(* Logix 5000 project; controller cal1615 1756-L62 rev 20.11; software revision 20.05; part 23 of 82 *)
(* tags used below, declared in another part *)
   FAULT : BOOL;   // Fault AFI
   HMI : BOOL;   // AFI HMI
   p01_sys_scp : SYS_SCP;   // System Scaling
   p01r02 : routine;   // System Misc Control
   p01r09_pb_global_reset : BOOL;   // System Modes PB: Global Fault Reset
   p12_ai_exhaust_amps : REAL;   // Zone 2 Analog Input Exhaust Fan Amps
   p12_ai_exhaust_hz : REAL;   // Zone 2 Analog Input Exhaust Fan HZ
   p12_ai_exhaust_hz_max : REAL;   // Zone 2 Analog Input Exhaust Fan Max HZ
   p12_ai_exhaust_rpm : REAL;   // Zone 2 Analog Input Exhaust Fan RPM
   p12_ai_lfl : REAL;   // Zone 2 Analog Input Lower Flash Limit
   p12_ai_prs : REAL;   // Zone 2 Analog Input Pressure
   p12_ai_recirc_amps : REAL;   // Zone 2 Analog Input Recirc Fan Amps
   p12_ai_recirc_hz : REAL;   // Zone 2 Analog Input Supply Fan HZ
   p12_ai_recirc_hz_max : REAL;   // Zone 2 Analog Input Supply Fan Max HZ
   p12_ai_recirc_rpm : REAL;   // Zone 2 Analog Input Recirc Fan RPM
   p12_ai_tc01 : REAL;   // Zone 2 Analog Input Control Thermocouple 1
   p12_ai_tc02 : REAL;   // Zone 2 Analog Input Control Thermocouple 2
   p12_ao_cv : REAL;   // Zone 2 Analog Output Control Valve
   p12_ao_exhaust_selected_speed : REAL;   // Zone 2 Analog Output Exhaust Fan VFD Selected Speed
   p12_ao_recirc_selected_speed : REAL;   // Zone 2 Analog Output Recirc Fan VFD Selected Speed
   p12_di_burner_auto : BOOL;   // Zone 2 Digital Input Burner Auto
   p12_di_burner_safeties_ok : BOOL;   // Zone 2 Digital Input Burner Safeties Ok
   p12_di_door_open : BOOL;   // Zone 2 Digital Input Access Door Open
   p12_di_exh : acs800_di_normal;   // Zone 2 Digital Inputs Exhaust Fan
   p12_di_exh_fan_mtr_ts : BOOL;   // Zone 2 Digital Input Exhaust Fan Motor Thermostat OK
   p12_di_exh_flow_ok : BOOL;   // Zone 2 Digital Input Exhaust Flow OK
   p12_di_flame_failure : BOOL;   // Zone 2 Digital Input Flame Failure
   p12_di_flame_on : BOOL;   // Zone 2 Digital Input Burner is On
   p12_di_fresh_air_clean : BOOL;   // Zone 2 Digital Input Fresh Air Filter Dirty
   p12_di_high_limit_temp_ok : BOOL;   // Zone 2 Digital Input High Limit Temperature OK
   p12_di_recirc : acs800_di_normal;   // Zone 2 Digital Inputs Recirc Fan
   p12_di_recirc_fan_mtr_ts : BOOL;   // Zone 2 Digital Input Recirc Fan Motor Thermostat OK
   p12_di_recirc_flow_ok : BOOL;   // Zone 2 Digital Input Recirc Flow OK
   p12_di_sp0 : BOOL;
   p12_di_sp00 : BOOL;   // Zone 2 Digital Input Combustion Blower Pressure OK
   p12_di_sp1 : BOOL;
   p12_di_sp2 : BOOL;
   p12_di_sp3 : BOOL;
   p12_di_tc01_bo : BOOL;   // Zone 2 Digital Input Control Thermocouple 1 Failure
   p12_di_tc02_bo : BOOL;   // Zone 2 Digital Input Control Thermocouple 2 Failure
   p12_di_zone_air_clean : BOOL;   // Zone 2 Digital Input Zone 2 Filter Dirty
   p12_dint_to_hmi : DINT[16];   // Zone 2 Temperature Control VFDs On
   p12_do_enable_burner : BOOL;   // Zone 2 Digital Output Enable Burner
   p12_do_exh : acs800_do_normal;   // Zone 2 Digital Output Exhaust Fan
   p12_do_recirc : acs800_do_normal;   // Zone 2 Digital Outputs Supply Fan
   p12_do_rst_flame : BOOL;   // Zone 2 Digital Output Reset Flame Safety
   p12_exhaust_input_max : REAL;
   p12_exhaust_input_min : REAL;
   p12_exhaust_output_max : REAL;
   p12_exhaust_output_min : REAL;
   p12_hc_input_max : REAL;
   p12_hc_input_min : REAL;
   p12_hc_output_max : REAL;
   p12_hc_output_min : REAL;
   p12_lfl_input_max : REAL;
   p12_lfl_input_min : REAL;
   p12_lfl_output_max : REAL;
   p12_lfl_output_min : REAL;
   p12_param_tc01z : REAL;   // Zone 2 Parameter Process Temperature Zero Offset
   p12_param_tc02z : REAL;   // Zone 2 Parameter SupplyTemperature Zero Offset
   p12_prs_input_max : REAL;
   p12_prs_input_min : REAL;
   p12_prs_output_max : REAL;
   p12_prs_output_min : REAL;
   p12_recirc_input_max : REAL;
   p12_recirc_input_min : REAL;
   p12_recirc_output_max : REAL;
   p12_recirc_output_min : REAL;
   p12r01 : routine;   // Zone 2 Main
   p12r03 : routine;   // Zone 2 Input
   p12r03_hz : SYS_SCP;   // Zone 2 Analog Inputs SCP Hz
   p12r03_timer_fault : TIMER[4];   // Zone 2 Input Fault Delay
   p12r03_timer_warning : TIMER[4];   // Zone 2 Input Warning Delay
   p12r04 : routine;   // Zone 2 Output
   p12r04_timer_fault : TIMER[4];   // Zone 2 Output Fault Delay
   p12r04_timer_warning : TIMER[4];   // Zone 2 Output Warning Delay
   p12r05 : routine;   // Zone 2 Dint to HMI
   p12r30 : routine;   // Zone 2 Temperature Control
   p12r30_request_heat : BOOL;   // Zone 2 Temperature Control Request Heat
   p12r30_request_manual : BOOL;   // Zone 2 Temperature Control Request Manual Control
   p12r30_vfds_ready : BOOL;   // Zone 2 Temperature Control VFDs On
   p12r31_request_auto_run : BOOL;   // Zone 2 Exhaust Fan Run Request
   p12r31_request_auto_stop : BOOL;   // Zone 2 Exhaust VFD Request Auto Stop
   p12r31_vfd_stopped : BOOL;   // Zone 2 Exhaust VFD VFD Stopped
   p12r32_request_auto_run : BOOL;   // Zone 2 Recirc Fan Run Request
   p12r32_request_auto_stop : BOOL;   // Zone 2 Recirc VFD Request Auto Stop
(* P12_Zone_2, continued *)

ROUTINE R03_Input   (* ladder *)
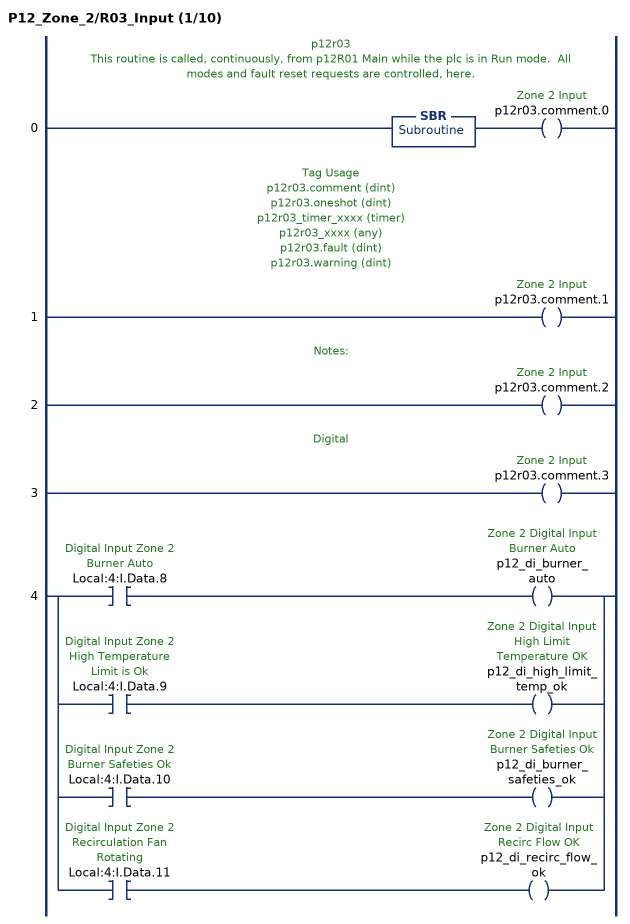
   // p12r03
   // This routine is called, continuously, from p12R01 Main while the plc is in Run mode.  All modes and fault reset requests are controlled, here.
   0: SBR()OTE(p12r03.comment.0);
   // Tag Usage
   // p12r03.comment (dint)
   // p12r03.oneshot (dint)
   // p12r03_timer_xxxx (timer)
   // p12r03_xxxx (any)
   // p12r03.fault (dint)
   // p12r03.warning (dint)
   1: OTE(p12r03.comment.1);
   // Notes:
   2: OTE(p12r03.comment.2);
   // Digital
   3: OTE(p12r03.comment.3);
   4: [XIC(Local:4:I.Data.8) OTE(p12_di_burner_auto) ,XIC(Local:4:I.Data.9) OTE(p12_di_high_limit_temp_ok) ,XIC(Local:4:I.Data.10) OTE(p12_di_burner_safeties_ok) ,XIC(Local:4:I.Data.11) OTE(p12_di_recirc_flow_ok) ];
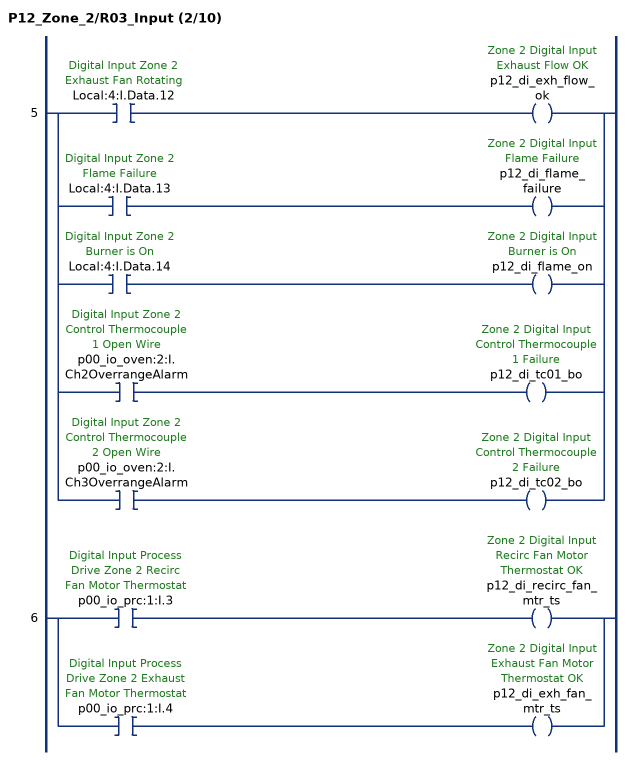
   5: [XIC(Local:4:I.Data.12) OTE(p12_di_exh_flow_ok) ,XIC(Local:4:I.Data.13) OTE(p12_di_flame_failure) ,XIC(Local:4:I.Data.14) OTE(p12_di_flame_on) ,XIC(p00_io_oven:2:I.Ch2OverrangeAlarm) OTE(p12_di_tc01_bo) ,XIC(p00_io_oven:2:I.Ch3OverrangeAlarm) OTE(p12_di_tc02_bo) ];
   6: [XIC(p00_io_prc:1:I.3) OTE(p12_di_recirc_fan_mtr_ts) ,XIC(p00_io_prc:1:I.4) OTE(p12_di_exh_fan_mtr_ts) ];
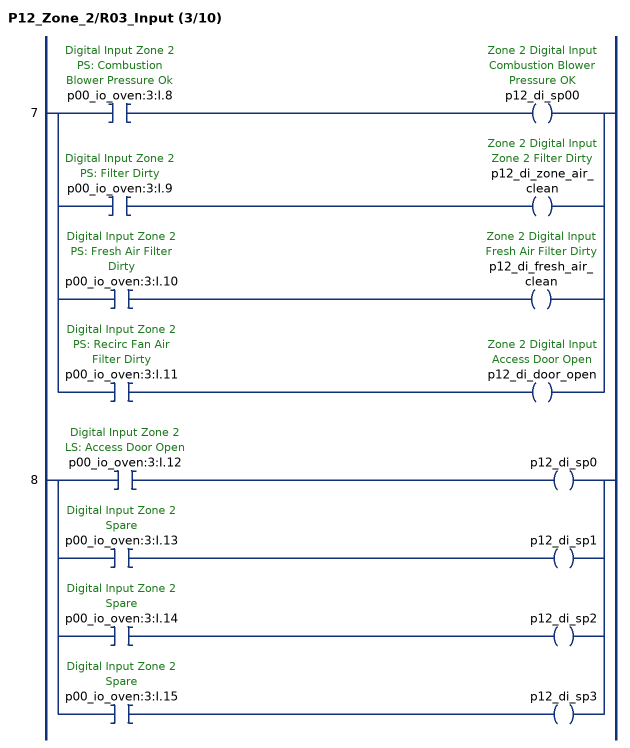
   7: [XIC(p00_io_oven:3:I.8) OTE(p12_di_sp00) ,XIC(p00_io_oven:3:I.9) OTE(p12_di_zone_air_clean) ,XIC(p00_io_oven:3:I.10) OTE(p12_di_fresh_air_clean) ,XIC(p00_io_oven:3:I.11) OTE(p12_di_door_open) ];
   8: [XIC(p00_io_oven:3:I.12) OTE(p12_di_sp0) ,XIC(p00_io_oven:3:I.13) OTE(p12_di_sp1) ,XIC(p00_io_oven:3:I.14) OTE(p12_di_sp2) ,XIC(p00_io_oven:3:I.15) OTE(p12_di_sp3) ];
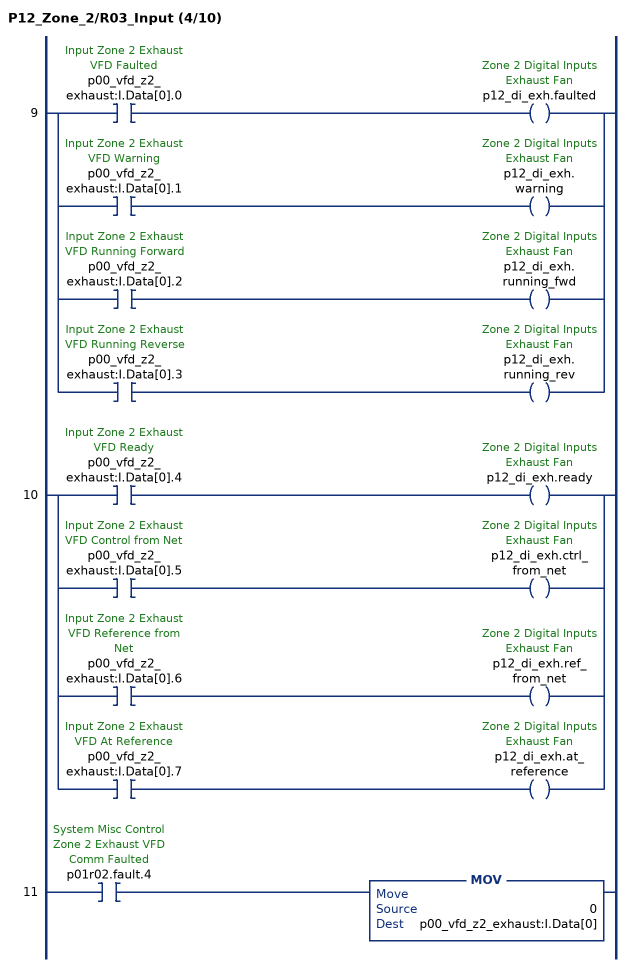
   9: [XIC(p00_vfd_z2_exhaust:I.Data[0].0) OTE(p12_di_exh.faulted) ,XIC(p00_vfd_z2_exhaust:I.Data[0].1) OTE(p12_di_exh.warning) ,XIC(p00_vfd_z2_exhaust:I.Data[0].2) OTE(p12_di_exh.running_fwd) ,XIC(p00_vfd_z2_exhaust:I.Data[0].3) OTE(p12_di_exh.running_rev) ];
   10: [XIC(p00_vfd_z2_exhaust:I.Data[0].4) OTE(p12_di_exh.ready) ,XIC(p00_vfd_z2_exhaust:I.Data[0].5) OTE(p12_di_exh.ctrl_from_net) ,XIC(p00_vfd_z2_exhaust:I.Data[0].6) OTE(p12_di_exh.ref_from_net) ,XIC(p00_vfd_z2_exhaust:I.Data[0].7) OTE(p12_di_exh.at_reference) ];
   11: XIC(p01r02.fault.4)MOV(0,p00_vfd_z2_exhaust:I.Data[0]);
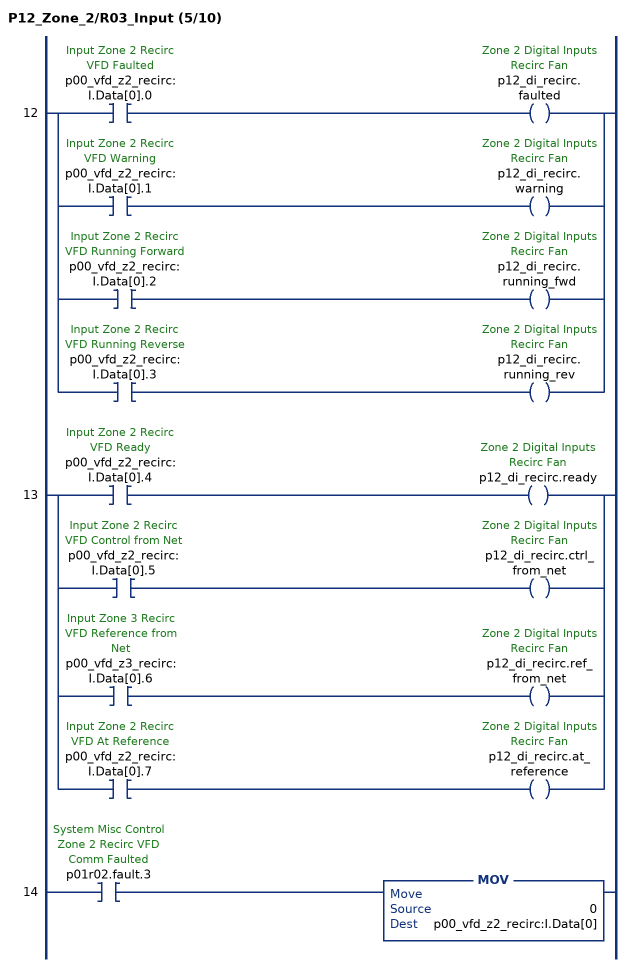
   12: [XIC(p00_vfd_z2_recirc:I.Data[0].0) OTE(p12_di_recirc.faulted) ,XIC(p00_vfd_z2_recirc:I.Data[0].1) OTE(p12_di_recirc.warning) ,XIC(p00_vfd_z2_recirc:I.Data[0].2) OTE(p12_di_recirc.running_fwd) ,XIC(p00_vfd_z2_recirc:I.Data[0].3) OTE(p12_di_recirc.running_rev) ];
   13: [XIC(p00_vfd_z2_recirc:I.Data[0].4) OTE(p12_di_recirc.ready) ,XIC(p00_vfd_z2_recirc:I.Data[0].5) OTE(p12_di_recirc.ctrl_from_net) ,XIC(p00_vfd_z3_recirc:I.Data[0].6) OTE(p12_di_recirc.ref_from_net) ,XIC(p00_vfd_z2_recirc:I.Data[0].7) OTE(p12_di_recirc.at_reference) ];
   14: XIC(p01r02.fault.3)MOV(0,p00_vfd_z2_recirc:I.Data[0]);
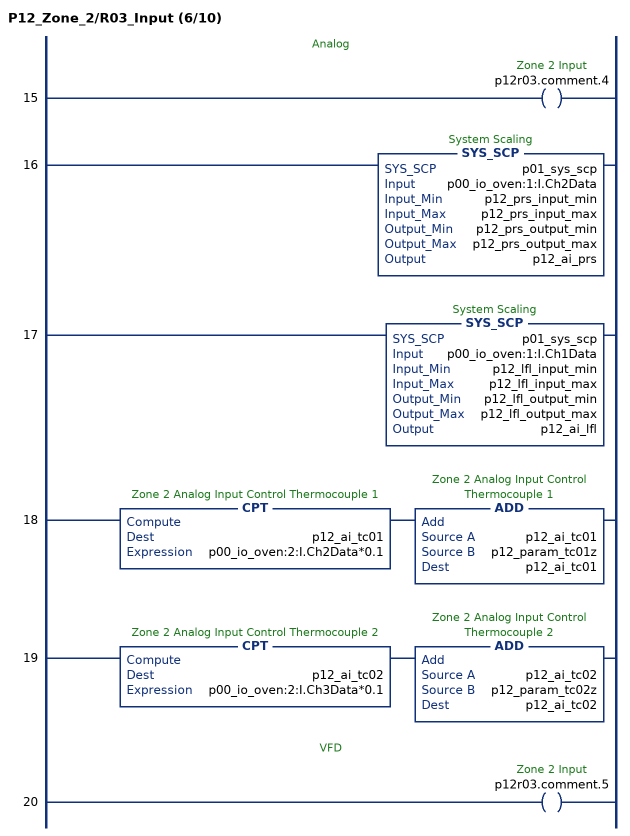
   // Analog
   15: OTE(p12r03.comment.4);
   16: SYS_SCP(p01_sys_scp,p00_io_oven:1:I.Ch2Data,p12_prs_input_min,p12_prs_input_max,p12_prs_output_min,p12_prs_output_max,p12_ai_prs);
   17: SYS_SCP(p01_sys_scp,p00_io_oven:1:I.Ch1Data,p12_lfl_input_min,p12_lfl_input_max,p12_lfl_output_min,p12_lfl_output_max,p12_ai_lfl);
   18: CPT(p12_ai_tc01,p00_io_oven:2:I.Ch2Data*0.1)ADD(p12_ai_tc01,p12_param_tc01z,p12_ai_tc01);
   19: CPT(p12_ai_tc02,p00_io_oven:2:I.Ch3Data*0.1)ADD(p12_ai_tc02,p12_param_tc02z,p12_ai_tc02);
   // VFD
   20: OTE(p12r03.comment.5);
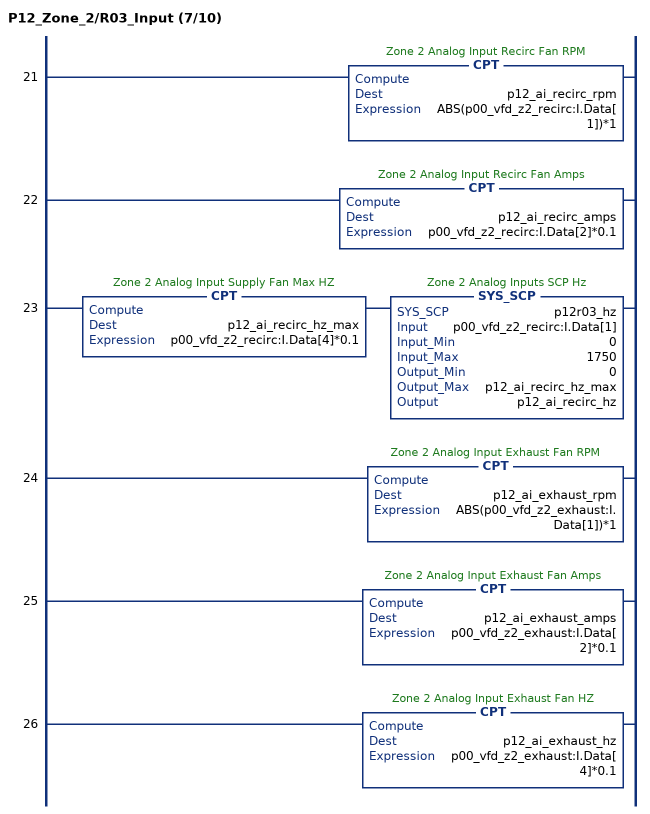
   21: CPT(p12_ai_recirc_rpm,ABS(p00_vfd_z2_recirc:I.Data[1])*1);
   22: CPT(p12_ai_recirc_amps,p00_vfd_z2_recirc:I.Data[2]*0.1);
   23: CPT(p12_ai_recirc_hz_max,p00_vfd_z2_recirc:I.Data[4]*0.1)SYS_SCP(p12r03_hz,p00_vfd_z2_recirc:I.Data[1],0,1750,0,p12_ai_recirc_hz_max,p12_ai_recirc_hz);
   24: CPT(p12_ai_exhaust_rpm,ABS(p00_vfd_z2_exhaust:I.Data[1])*1);
   25: CPT(p12_ai_exhaust_amps,p00_vfd_z2_exhaust:I.Data[2]*0.1);
   26: CPT(p12_ai_exhaust_hz,p00_vfd_z2_exhaust:I.Data[4]*0.1);
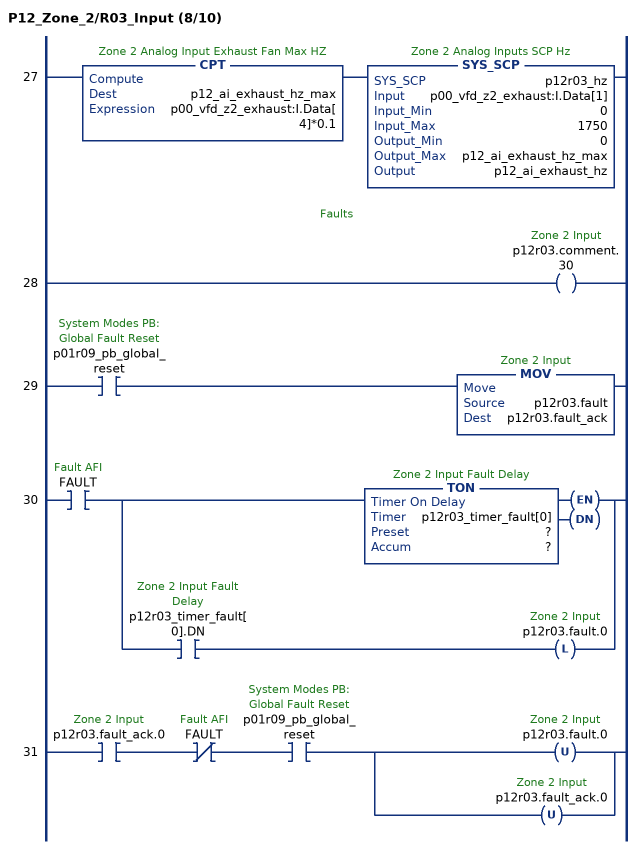
   27: CPT(p12_ai_exhaust_hz_max,p00_vfd_z2_exhaust:I.Data[4]*0.1)SYS_SCP(p12r03_hz,p00_vfd_z2_exhaust:I.Data[1],0,1750,0,p12_ai_exhaust_hz_max,p12_ai_exhaust_hz);
   // Faults
   28: OTE(p12r03.comment.30);
   29: XIC(p01r09_pb_global_reset)MOV(p12r03.fault,p12r03.fault_ack);
   30: XIC(FAULT)[TON(p12r03_timer_fault[0],?,?) ,XIC(p12r03_timer_fault[0].DN) OTL(p12r03.fault.0) ];
   31: XIC(p12r03.fault_ack.0)XIO(FAULT)XIC(p01r09_pb_global_reset)[OTU(p12r03.fault.0) ,OTU(p12r03.fault_ack.0) ];
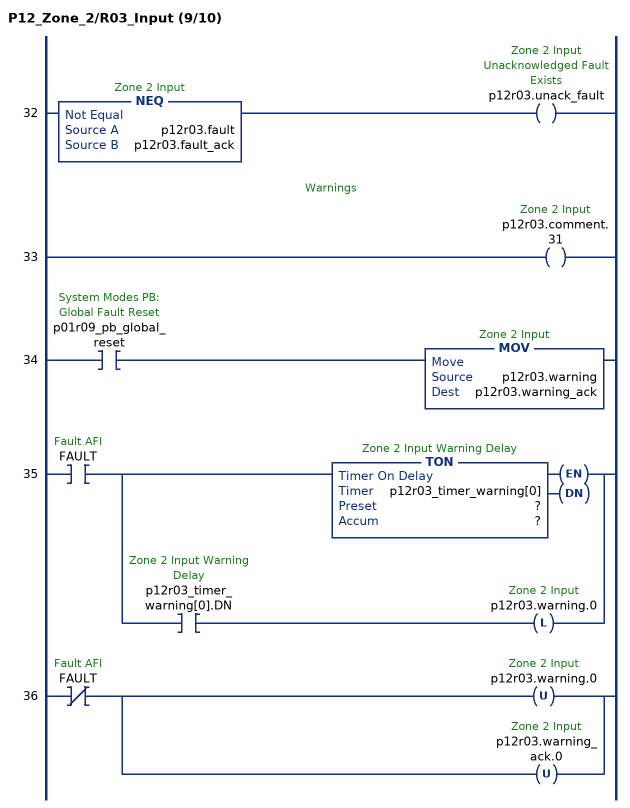
   32: NEQ(p12r03.fault,p12r03.fault_ack)OTE(p12r03.unack_fault);
   // Warnings
   33: OTE(p12r03.comment.31);
   34: XIC(p01r09_pb_global_reset)MOV(p12r03.warning,p12r03.warning_ack);
   35: XIC(FAULT)[TON(p12r03_timer_warning[0],?,?) ,XIC(p12r03_timer_warning[0].DN) OTL(p12r03.warning.0) ];
   36: XIO(FAULT)[OTU(p12r03.warning.0) ,OTU(p12r03.warning_ack.0) ];
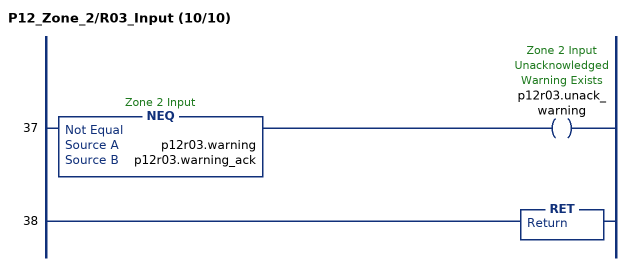
   37: NEQ(p12r03.warning,p12r03.warning_ack)OTE(p12r03.unack_warning);
   38: RET();
END_ROUTINE

ROUTINE R04_Output   (* ladder *)
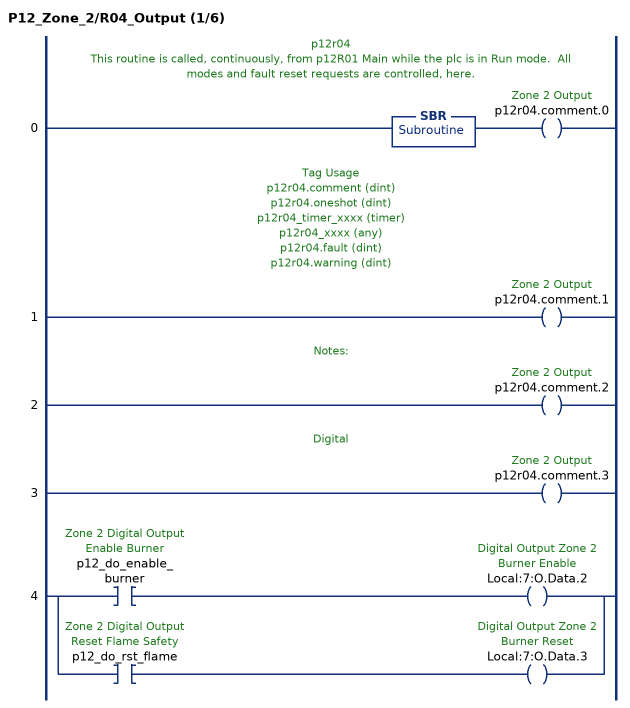
   // p12r04
   // This routine is called, continuously, from p12R01 Main while the plc is in Run mode.  All modes and fault reset requests are controlled, here.
   0: SBR()OTE(p12r04.comment.0);
   // Tag Usage
   // p12r04.comment (dint)
   // p12r04.oneshot (dint)
   // p12r04_timer_xxxx (timer)
   // p12r04_xxxx (any)
   // p12r04.fault (dint)
   // p12r04.warning (dint)
   1: OTE(p12r04.comment.1);
   // Notes:
   2: OTE(p12r04.comment.2);
   // Digital
   3: OTE(p12r04.comment.3);
   4: [XIC(p12_do_enable_burner) OTE(Local:7:O.Data.2) ,XIC(p12_do_rst_flame) OTE(Local:7:O.Data.3) ];
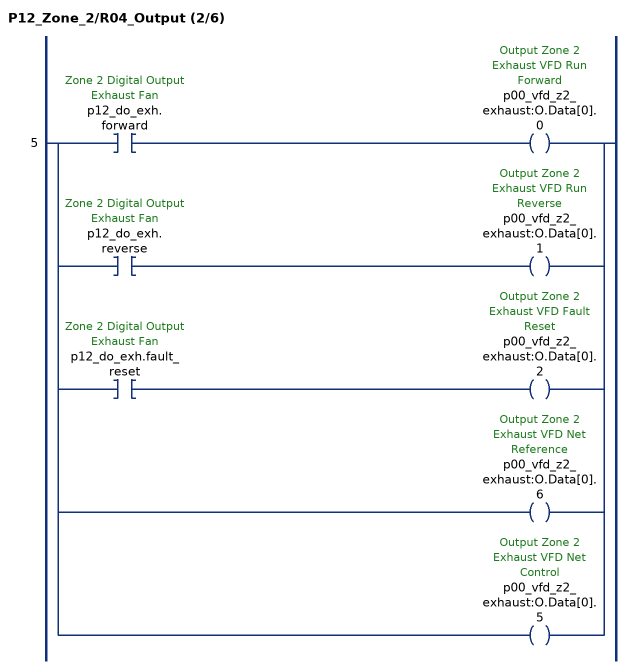
   5: [XIC(p12_do_exh.forward) OTE(p00_vfd_z2_exhaust:O.Data[0].0) ,XIC(p12_do_exh.reverse) OTE(p00_vfd_z2_exhaust:O.Data[0].1) ,XIC(p12_do_exh.fault_reset) OTE(p00_vfd_z2_exhaust:O.Data[0].2) ,OTE(p00_vfd_z2_exhaust:O.Data[0].6) ,OTE(p00_vfd_z2_exhaust:O.Data[0].5) ];
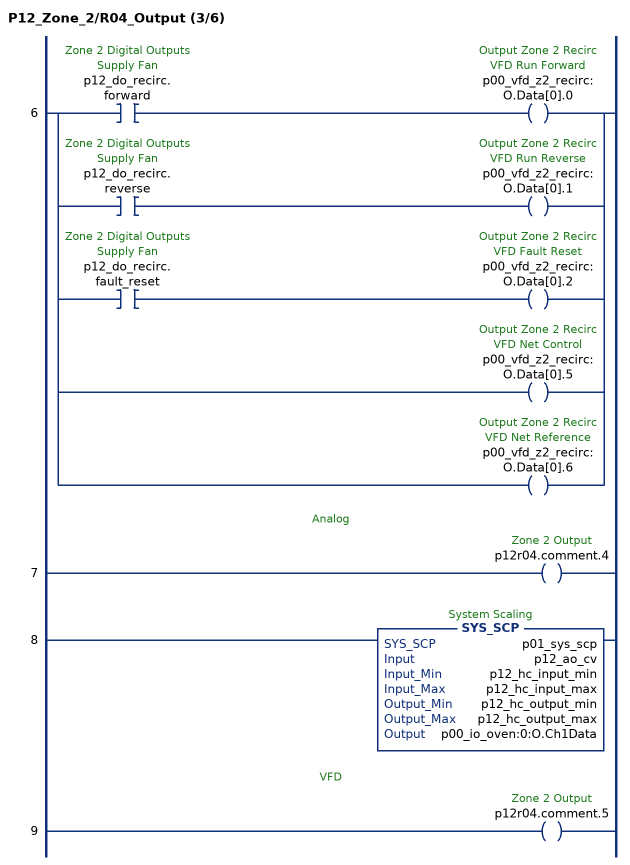
   6: [XIC(p12_do_recirc.forward) OTE(p00_vfd_z2_recirc:O.Data[0].0) ,XIC(p12_do_recirc.reverse) OTE(p00_vfd_z2_recirc:O.Data[0].1) ,XIC(p12_do_recirc.fault_reset) OTE(p00_vfd_z2_recirc:O.Data[0].2) ,OTE(p00_vfd_z2_recirc:O.Data[0].5) ,OTE(p00_vfd_z2_recirc:O.Data[0].6) ];
   // Analog
   7: OTE(p12r04.comment.4);
   8: SYS_SCP(p01_sys_scp,p12_ao_cv,p12_hc_input_min,p12_hc_input_max,p12_hc_output_min,p12_hc_output_max,p00_io_oven:0:O.Ch1Data);
   // VFD
   9: OTE(p12r04.comment.5);
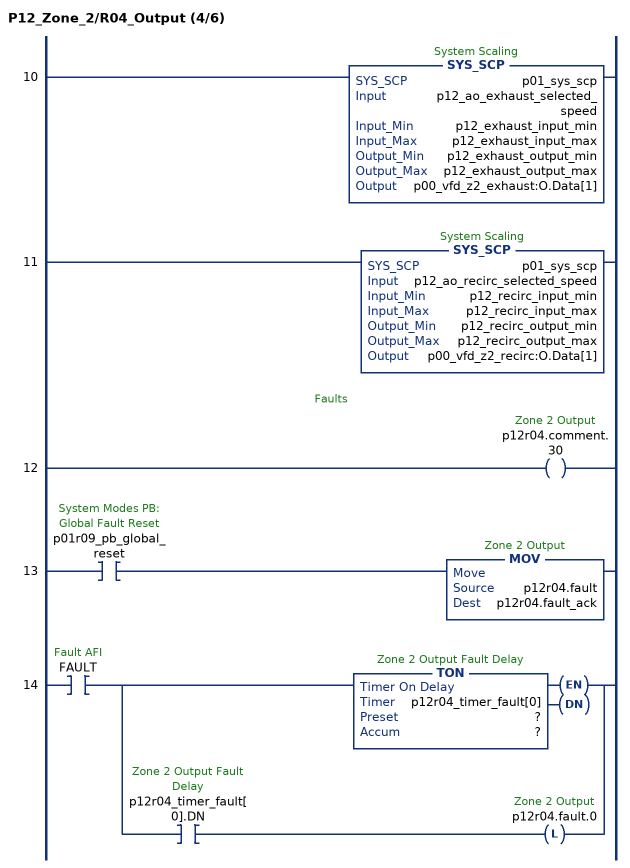
   10: SYS_SCP(p01_sys_scp,p12_ao_exhaust_selected_speed,p12_exhaust_input_min,p12_exhaust_input_max,p12_exhaust_output_min,p12_exhaust_output_max,p00_vfd_z2_exhaust:O.Data[1]);
   11: SYS_SCP(p01_sys_scp,p12_ao_recirc_selected_speed,p12_recirc_input_min,p12_recirc_input_max,p12_recirc_output_min,p12_recirc_output_max,p00_vfd_z2_recirc:O.Data[1]);
   // Faults
   12: OTE(p12r04.comment.30);
   13: XIC(p01r09_pb_global_reset)MOV(p12r04.fault,p12r04.fault_ack);
   14: XIC(FAULT)[TON(p12r04_timer_fault[0],?,?) ,XIC(p12r04_timer_fault[0].DN) OTL(p12r04.fault.0) ];
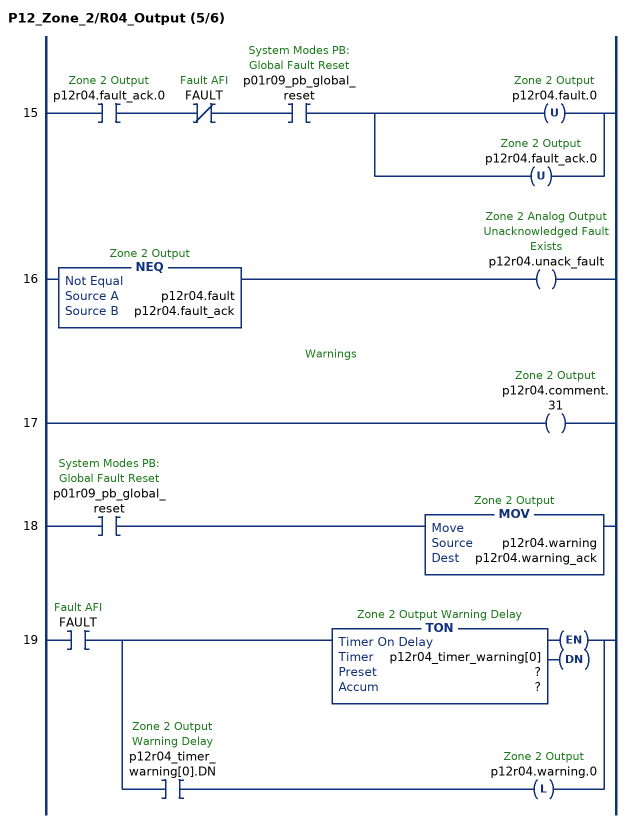
   15: XIC(p12r04.fault_ack.0)XIO(FAULT)XIC(p01r09_pb_global_reset)[OTU(p12r04.fault.0) ,OTU(p12r04.fault_ack.0) ];
   16: NEQ(p12r04.fault,p12r04.fault_ack)OTE(p12r04.unack_fault);
   // Warnings
   17: OTE(p12r04.comment.31);
   18: XIC(p01r09_pb_global_reset)MOV(p12r04.warning,p12r04.warning_ack);
   19: XIC(FAULT)[TON(p12r04_timer_warning[0],?,?) ,XIC(p12r04_timer_warning[0].DN) OTL(p12r04.warning.0) ];
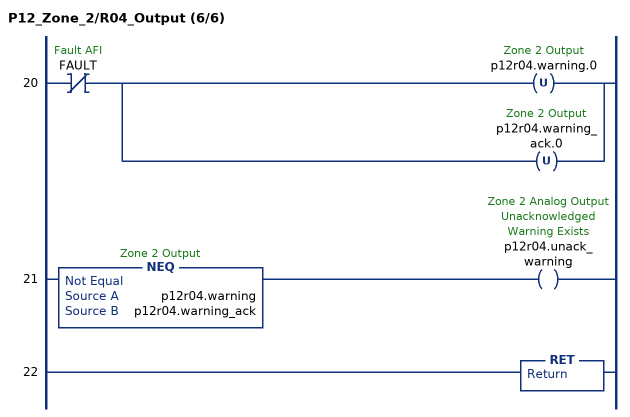
   20: XIO(FAULT)[OTU(p12r04.warning.0) ,OTU(p12r04.warning_ack.0) ];
   21: NEQ(p12r04.warning,p12r04.warning_ack)OTE(p12r04.unack_warning);
   22: RET();
END_ROUTINE

ROUTINE R05_Dint_to_HMI   (* ladder *)
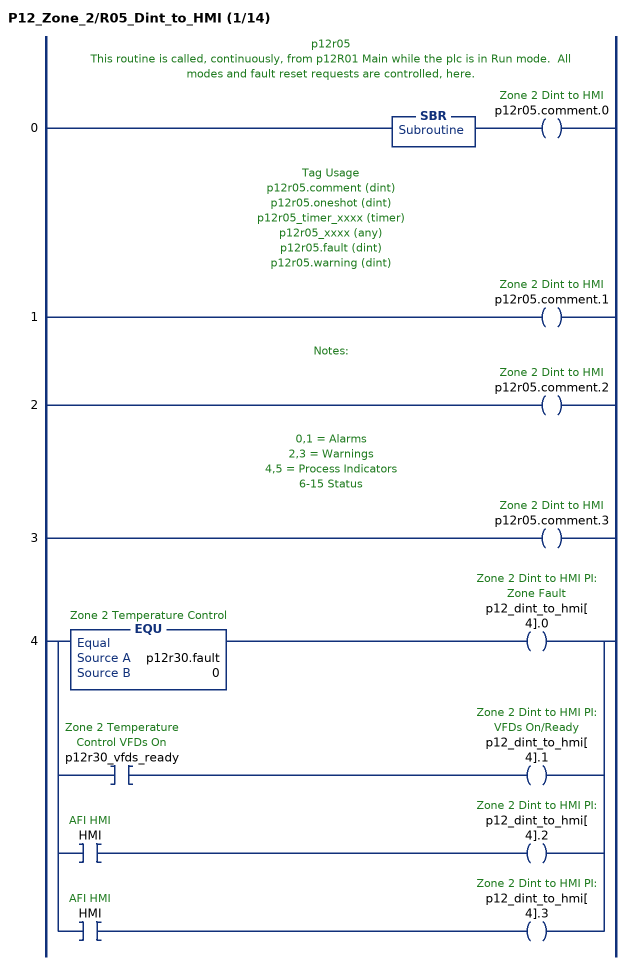
   // p12r05
   // This routine is called, continuously, from p12R01 Main while the plc is in Run mode.  All modes and fault reset requests are controlled, here.
   0: SBR()OTE(p12r05.comment.0);
   // Tag Usage
   // p12r05.comment (dint)
   // p12r05.oneshot (dint)
   // p12r05_timer_xxxx (timer)
   // p12r05_xxxx (any)
   // p12r05.fault (dint)
   // p12r05.warning (dint)
   1: OTE(p12r05.comment.1);
   // Notes:
   2: OTE(p12r05.comment.2);
   // 0,1 = Alarms
   // 2,3 = Warnings
   // 4,5 = Process Indicators
   // 6-15 Status
   3: OTE(p12r05.comment.3);
   4: [EQU(p12r30.fault,0) OTE(p12_dint_to_hmi[4].0) ,XIC(p12r30_vfds_ready) OTE(p12_dint_to_hmi[4].1) ,XIC(HMI) OTE(p12_dint_to_hmi[4].2) ,XIC(HMI) OTE(p12_dint_to_hmi[4].3) ];
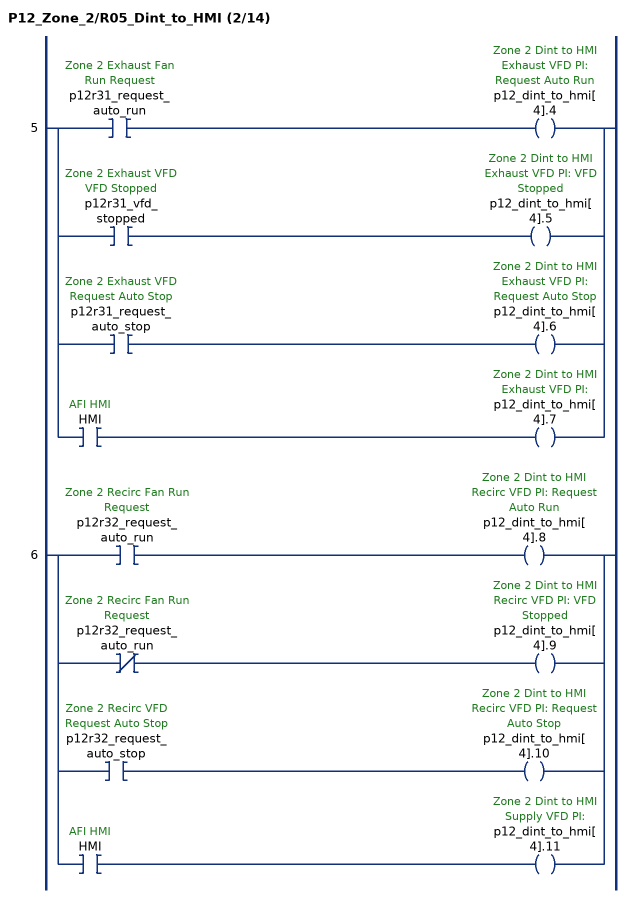
   5: [XIC(p12r31_request_auto_run) OTE(p12_dint_to_hmi[4].4) ,XIC(p12r31_vfd_stopped) OTE(p12_dint_to_hmi[4].5) ,XIC(p12r31_request_auto_stop) OTE(p12_dint_to_hmi[4].6) ,XIC(HMI) OTE(p12_dint_to_hmi[4].7) ];
   6: [XIC(p12r32_request_auto_run) OTE(p12_dint_to_hmi[4].8) ,XIO(p12r32_request_auto_run) OTE(p12_dint_to_hmi[4].9) ,XIC(p12r32_request_auto_stop) OTE(p12_dint_to_hmi[4].10) ,XIC(HMI) OTE(p12_dint_to_hmi[4].11) ];
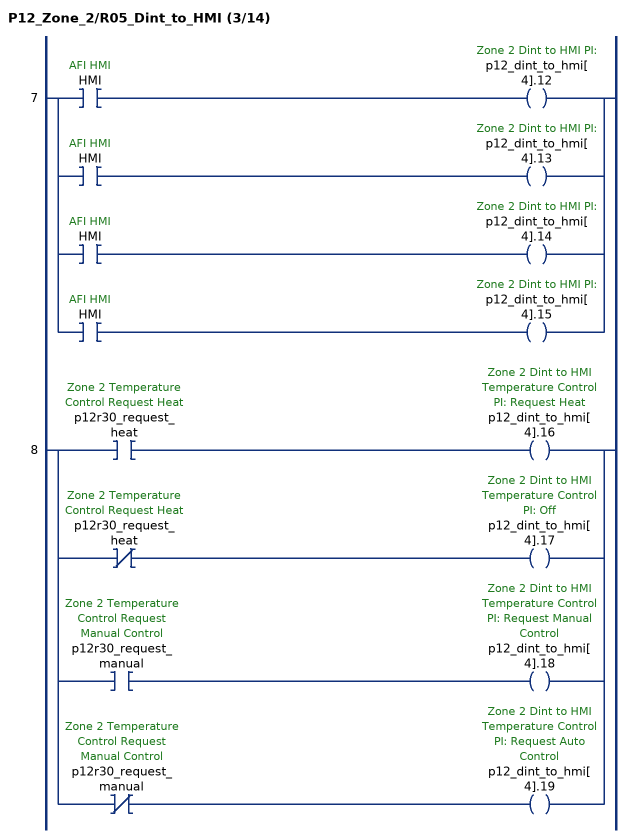
   7: [XIC(HMI) OTE(p12_dint_to_hmi[4].12) ,XIC(HMI) OTE(p12_dint_to_hmi[4].13) ,XIC(HMI) OTE(p12_dint_to_hmi[4].14) ,XIC(HMI) OTE(p12_dint_to_hmi[4].15) ];
   8: [XIC(p12r30_request_heat) OTE(p12_dint_to_hmi[4].16) ,XIO(p12r30_request_heat) OTE(p12_dint_to_hmi[4].17) ,XIC(p12r30_request_manual) OTE(p12_dint_to_hmi[4].18) ,XIO(p12r30_request_manual) OTE(p12_dint_to_hmi[4].19) ];
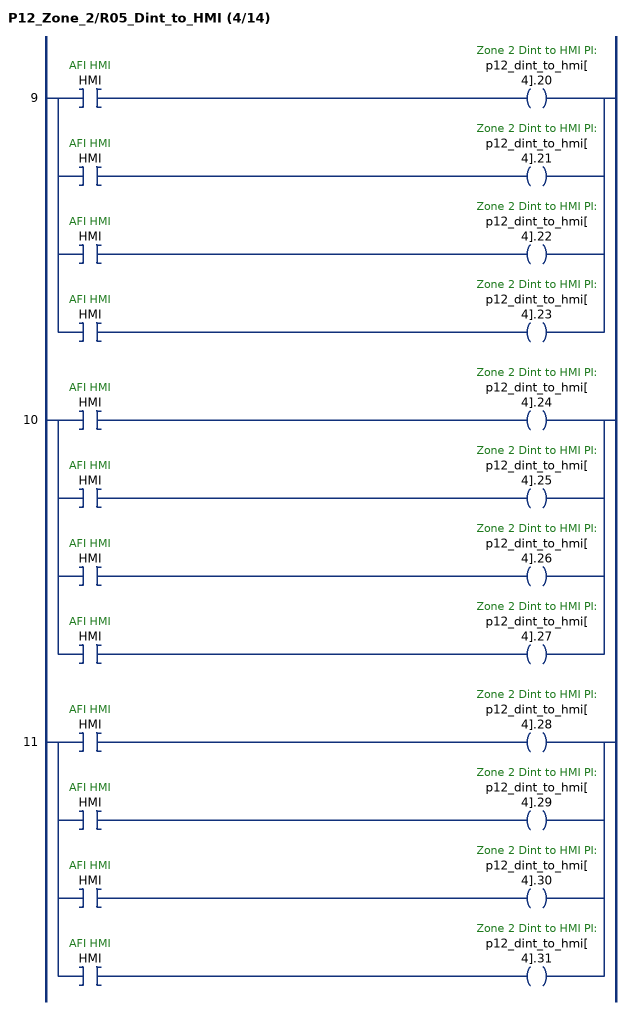
   9: [XIC(HMI) OTE(p12_dint_to_hmi[4].20) ,XIC(HMI) OTE(p12_dint_to_hmi[4].21) ,XIC(HMI) OTE(p12_dint_to_hmi[4].22) ,XIC(HMI) OTE(p12_dint_to_hmi[4].23) ];
   10: [XIC(HMI) OTE(p12_dint_to_hmi[4].24) ,XIC(HMI) OTE(p12_dint_to_hmi[4].25) ,XIC(HMI) OTE(p12_dint_to_hmi[4].26) ,XIC(HMI) OTE(p12_dint_to_hmi[4].27) ];
   11: [XIC(HMI) OTE(p12_dint_to_hmi[4].28) ,XIC(HMI) OTE(p12_dint_to_hmi[4].29) ,XIC(HMI) OTE(p12_dint_to_hmi[4].30) ,XIC(HMI) OTE(p12_dint_to_hmi[4].31) ];
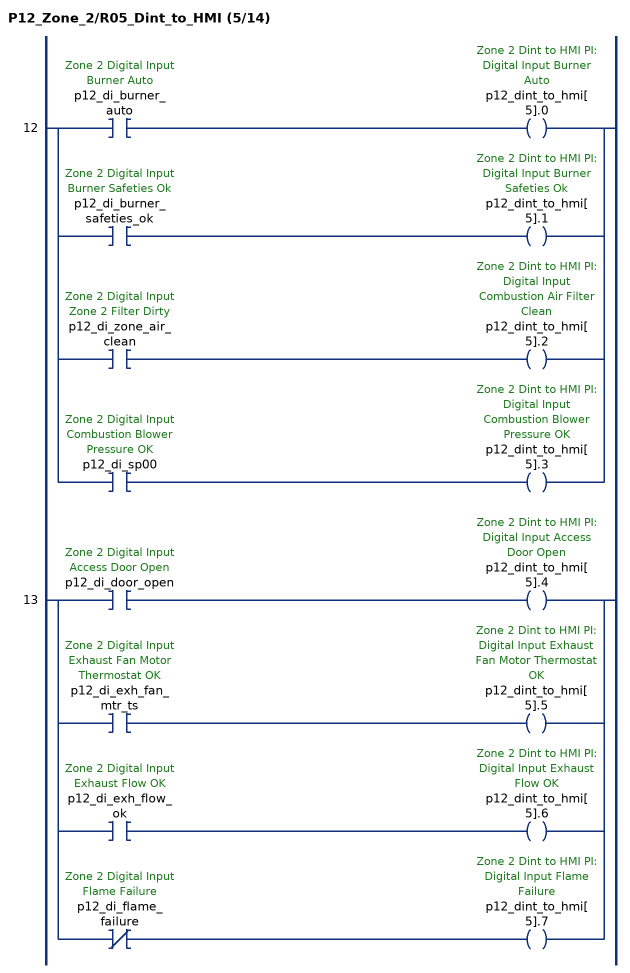
   12: [XIC(p12_di_burner_auto) OTE(p12_dint_to_hmi[5].0) ,XIC(p12_di_burner_safeties_ok) OTE(p12_dint_to_hmi[5].1) ,XIC(p12_di_zone_air_clean) OTE(p12_dint_to_hmi[5].2) ,XIC(p12_di_sp00) OTE(p12_dint_to_hmi[5].3) ];
   13: [XIC(p12_di_door_open) OTE(p12_dint_to_hmi[5].4) ,XIC(p12_di_exh_fan_mtr_ts) OTE(p12_dint_to_hmi[5].5) ,XIC(p12_di_exh_flow_ok) OTE(p12_dint_to_hmi[5].6) ,XIO(p12_di_flame_failure) OTE(p12_dint_to_hmi[5].7) ];
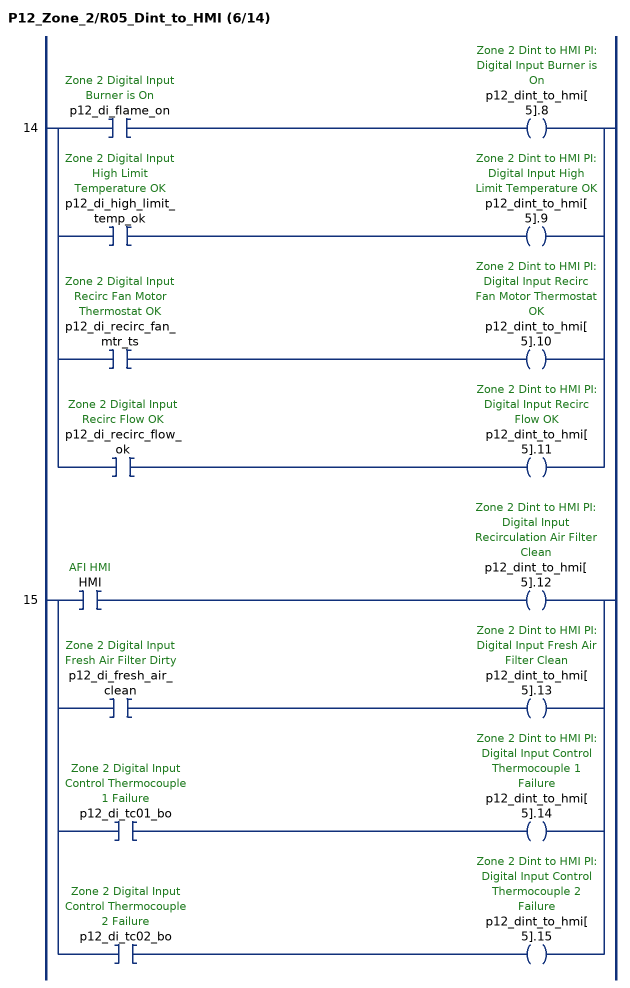
   14: [XIC(p12_di_flame_on) OTE(p12_dint_to_hmi[5].8) ,XIC(p12_di_high_limit_temp_ok) OTE(p12_dint_to_hmi[5].9) ,XIC(p12_di_recirc_fan_mtr_ts) OTE(p12_dint_to_hmi[5].10) ,XIC(p12_di_recirc_flow_ok) OTE(p12_dint_to_hmi[5].11) ];
   15: [XIC(HMI) OTE(p12_dint_to_hmi[5].12) ,XIC(p12_di_fresh_air_clean) OTE(p12_dint_to_hmi[5].13) ,XIC(p12_di_tc01_bo) OTE(p12_dint_to_hmi[5].14) ,XIC(p12_di_tc02_bo) OTE(p12_dint_to_hmi[5].15) ];
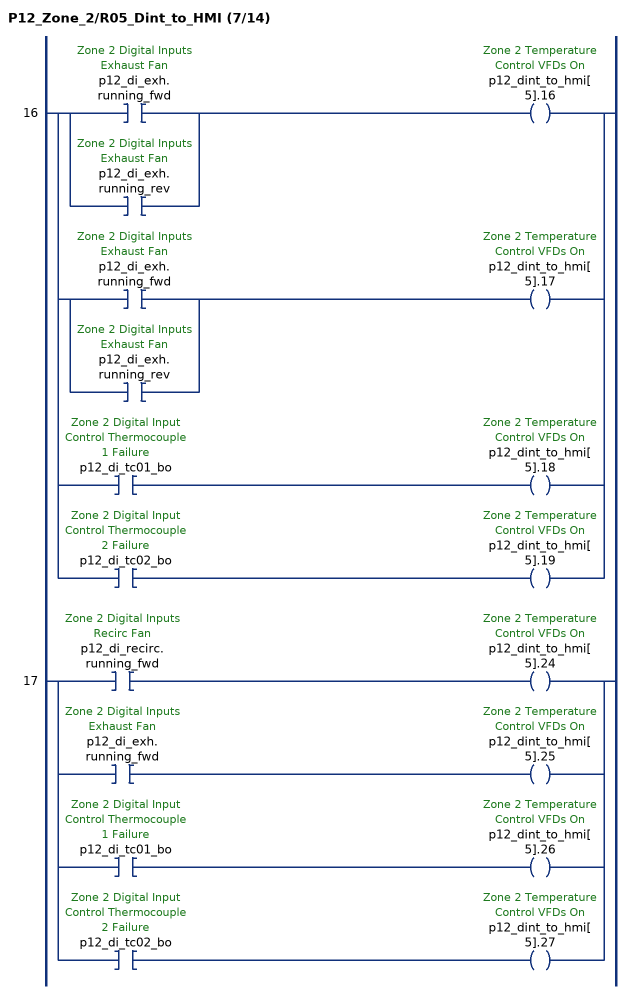
   16: [[XIC(p12_di_exh.running_fwd) ,XIC(p12_di_exh.running_rev) ] OTE(p12_dint_to_hmi[5].16) ,[XIC(p12_di_exh.running_fwd) ,XIC(p12_di_exh.running_rev) ] OTE(p12_dint_to_hmi[5].17) ,XIC(p12_di_tc01_bo) OTE(p12_dint_to_hmi[5].18) ,XIC(p12_di_tc02_bo) OTE(p12_dint_to_hmi[5].19) ];
   17: [XIC(p12_di_recirc.running_fwd) OTE(p12_dint_to_hmi[5].24) ,XIC(p12_di_exh.running_fwd) OTE(p12_dint_to_hmi[5].25) ,XIC(p12_di_tc01_bo) OTE(p12_dint_to_hmi[5].26) ,XIC(p12_di_tc02_bo) OTE(p12_dint_to_hmi[5].27) ];
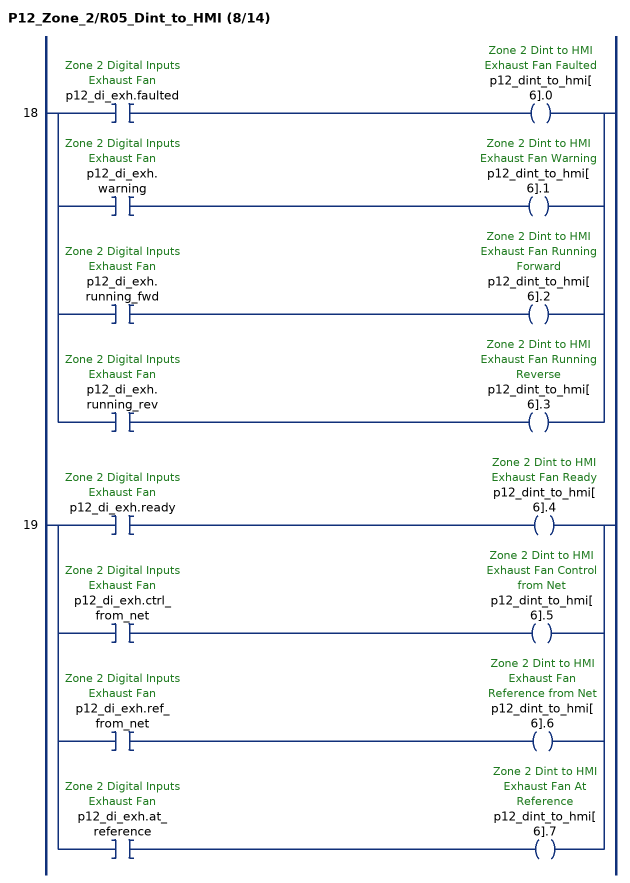
   18: [XIC(p12_di_exh.faulted) OTE(p12_dint_to_hmi[6].0) ,XIC(p12_di_exh.warning) OTE(p12_dint_to_hmi[6].1) ,XIC(p12_di_exh.running_fwd) OTE(p12_dint_to_hmi[6].2) ,XIC(p12_di_exh.running_rev) OTE(p12_dint_to_hmi[6].3) ];
   19: [XIC(p12_di_exh.ready) OTE(p12_dint_to_hmi[6].4) ,XIC(p12_di_exh.ctrl_from_net) OTE(p12_dint_to_hmi[6].5) ,XIC(p12_di_exh.ref_from_net) OTE(p12_dint_to_hmi[6].6) ,XIC(p12_di_exh.at_reference) OTE(p12_dint_to_hmi[6].7) ];
